(*
version 1.0	21 feb 2008
programmer 	hugo
tested by	oscat

this function multiplies two complex numbers

*)
FUNCTION CMUL : complex
VAR_INPUT
	X, Y : complex;
END_VAR

CMUL.re := X.re * Y.re - X.im * Y.im;
CMUL.im := X.re * Y.im + X.im * Y.re;

(* revision history
hm	21. feb 2008	rev 1.0
	original version

*)

END_FUNCTION

(* stored: Version 1.1.0.1
   POU CMUL: Id {dc265928-fff5-4a1a-9b05-e47e70b1396a}, SpecialFunc None *)
